(* Schneider Machine Expert - Basic project automated sorting system, file version 2.7.0.0 *)
(* ProjectInformations: Name=New project *)

HARDWARE
  Cpu 0: TM221M16R/G
  EthernetConfiguration: NetworkName=M221, IpAllocationMode=FixedAddress, IpAddress=0.0.0.0, SubnetMask=0.0.0.0
  SerialLineConfiguration: Baud=Baud19200, Parity=ParityEven, DataBits=DataBits8, StopBits=StopBits1, PhysicalMedium=PhysicalMediumRs485, TransmissionMode=TransmissionModeModbusRtu, SlaveId=1, Addressing=SlaveAddressing
  MastTask: UsePeriodScanMode=false, PeriodScan=100
  FastTask: Period=255
  CpuBehavior: StartingMode=StartAsPreviousState, AutoSaveRamOnEeprom=true, WatchdogPeriod=250

SYMBOLS  (address, symbol, comment, settings)
  %I0.0     IS_WOOD
  %I0.1     IS_PLASTIC
  %I0.2     IS_METAL
  %Q0.0     SORT_TO_WOOD
  %Q0.1     SORT_TO_PLASTIC
  %Q0.2     SORT_TO_METAL
  %Q0.3     CONVEYORT

POU New POU
  (* SectionNumber=0 *)

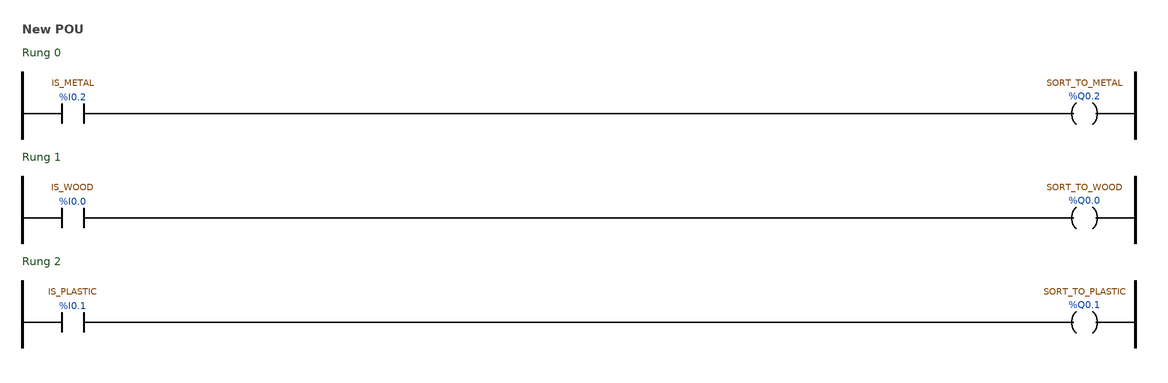

// Rung 0
  LD %I0.2                (* IS_METAL *)
  ST %Q0.2                (* SORT_TO_METAL *)
  // as ST:
  //   SORT_TO_METAL := IS_METAL;

// Rung 1
  LD %I0.0                (* IS_WOOD *)
  ST %Q0.0                (* SORT_TO_WOOD *)
  // as ST:
  //   SORT_TO_WOOD := IS_WOOD;

// Rung 2
  LD %I0.1                (* IS_PLASTIC *)
  ST %Q0.1                (* SORT_TO_PLASTIC *)
  // as ST:
  //   SORT_TO_PLASTIC := IS_PLASTIC;
